// TIA Portal V17 export
// export: Created 2023-02-13T11:16:40.304202Z, ExportSetting WithDefaults, DisplayName Totally Integrated Automation Portal, DisplayVersion V17, DisplayName TIA Portal Openness, DisplayVersion V17, DisplayName TIA Portal Teamcenter Gateway, DisplayVersion V17, DisplayName TIA Portal Version Control Interface, DisplayVersion V17, DisplayName SINAMICS Startdrive Advanced, DisplayVersion V17, DisplayName SINAMICS Startdrive G130, G150, S120, S150, SINAMICS MV, S210, DisplayVersion V17, DisplayName SINAMICS Startdrive G110M, G120, G120C, G120D, G120P, G115D, DisplayVersion V17, DisplayName STEP 7 Professional, DisplayVersion V17, DisplayName STEP 7 Safety, DisplayVersion V17, DisplayName WinCC Professional, DisplayVersion V17
FUNCTION_BLOCK "Hot_Water"   // FB366, LAD
{ S7_Optimized_Access := 'TRUE' }
VERSION : 0.1
// stored: AutoNumber false, IsIECCheckEnabled false, IsRetainMemResEnabled false, MemoryReserve 100, SetENOAutomatically false, UDAEnableTagReadback false
   VAR_INPUT
      IN_FBAV_Inload : Bool;
      IN_FBAV_Outlet : Bool;
      IN_FBAV_Transfer : Bool;
      IN_FBP_Transfer : Bool;
      IN_FBP_Transfer_SP : Real;
      IN_Dose_Run : Bool;
      IN_Dose_Held : Bool;
      IN_Dose_Complete : Bool;
      IN_Dose_Header_1 : Bool;
      IN_Dose_Header_2 : Bool;
      IN_Dose_Valve_Cmd : Bool;
      IN_Dose_Pump_Cmd : Bool;
      IN_Dose_Pump_Sp : Real;
      IN_Dose_LineOK : Bool;
      IN_Low_Level : Bool;
      IN_Med_Level : Bool;
      IN_High_Level : Bool;
      IN_FBCV : Bool;
      "IN_FBCV_Act%" : Real;
      IN_Temperature : Real;
   END_VAR
   VAR_OUTPUT
      Out_AV_Inload : Bool;
      Out_AV_Outlet : Bool;
      Out_AV_Transfer : Bool;
      Out_P_Transfer : Bool;
      Out_P_Transfer_Sp : Real;
      OUT_CV : Bool;
      Out_Temp_Act : Real;
      Out_Temp_Sp : Real;
   END_VAR
   VAR
      Cmd : Struct
         Inload_Start : Bool;
         Inload_Mode : Bool := 1;   // 0 : Manual ;; 1 : Auto
         ReadyForTransfer : Bool;
         Transfer_Mode : Bool;   // 0 : By Timer ;; 1 : By Quantity
      END_STRUCT;
   END_VAR
   VAR RETAIN
      Param : Struct
         Temperature_SP : Real := 50.0;
      END_STRUCT;
   END_VAR
   VAR
      State : Struct
         Tank_LL : Bool;
         Tank_ML : Bool;
         Tank_HL : Bool;
         Inload_EN : Bool;
         Inload_Aut : Bool;
         Inloading : Bool;
         Ready_For_Transfer_EN : Bool;
         Ready_For_Transfer : Bool;
         Tank_Available : Bool;
         Transfer_on_Prog : Bool;
      END_STRUCT;
      alwaysON : Bool;
      r : Struct
         PosE1 : Bool;
         PosE2 : Bool;
         PosE3 : Bool;
         PosE4 : Bool;
         PosE5 : Bool;
         PosE6 : Bool;
         PosE7 : Bool;
         PosE8 : Bool;
         PosE9 : Bool;
         PosE10 : Bool;
         PosE11 : Bool;
         PosE12 : Bool;
         PosE13 : Bool;
         PosE14 : Bool;
         PosE15 : Bool;
         PosE16 : Bool;
         PosE17 : Bool;
         PosE18 : Bool;
         PosE19 : Bool;
         PosE20 : Bool;
         PosE21 : Bool;
         PosE22 : Bool;
         PosE23 : Bool;
         PosE24 : Bool;
         PosE25 : Bool;
         PosE26 : Bool;
         PosE27 : Bool;
         PosE28 : Bool;
         PosE29 : Bool;
         PosE30 : Bool;
         PosE31 : Bool;
         PosE32 : Bool;
      END_STRUCT;
      Actuator : Struct
         AV_Inload : Bool;
         AV_Outlet : Bool;
         AV_Transfer : Bool;
         AV_CIP_Tank : Bool;
         AV_CIP_Line : Bool;
         P_Transfer : Bool;
         P_Inload : Bool;
         P_CIP : Bool;
         CV : Bool;
      END_STRUCT;
      SPumpTim { S7_SetPoint := 'True'} : TON_TIME;
   END_VAR
   VAR_TEMP   // added for the SCL form of the ladder/FBD networks
      _w1 : Bool;
      _w2 : Bool;
   END_VAR
BEGIN

REGION Network 1: Always_ON
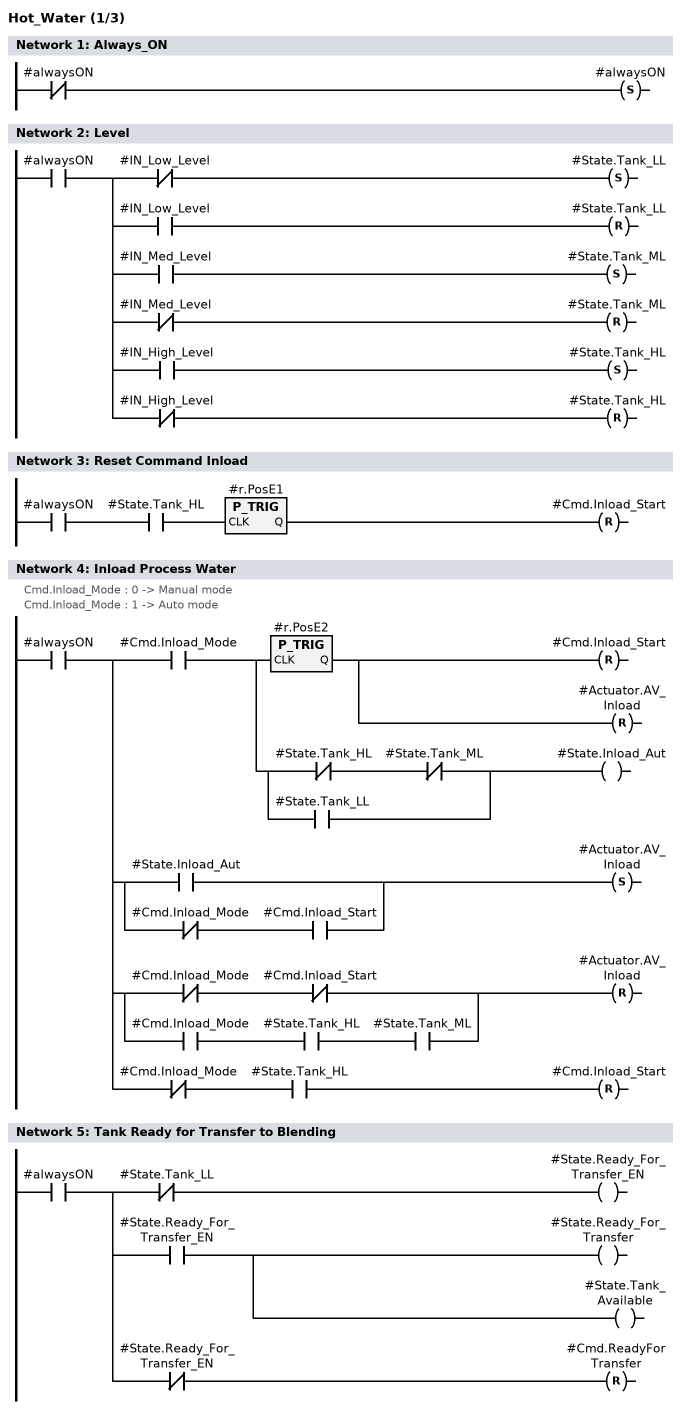
   RUNG wire#powerrail
      I_Contact( #alwaysON )
      S_Coil( #alwaysON )
   END_RUNG
   // the same network as SCL:
   IF NOT #alwaysON THEN #alwaysON := TRUE; END_IF;
END_REGION

REGION Network 2: Level
   RUNG wire#powerrail
      Contact( #alwaysON )
      wire#w1
      I_Contact( #IN_Low_Level )
      S_Coil( #State.Tank_LL )
   END_RUNG
   RUNG wire#w1
      Contact( #IN_Low_Level )
      R_Coil( #State.Tank_LL )
   END_RUNG
   RUNG wire#w1
      Contact( #IN_Med_Level )
      S_Coil( #State.Tank_ML )
   END_RUNG
   RUNG wire#w1
      I_Contact( #IN_Med_Level )
      R_Coil( #State.Tank_ML )
   END_RUNG
   RUNG wire#w1
      Contact( #IN_High_Level )
      S_Coil( #State.Tank_HL )
   END_RUNG
   RUNG wire#w1
      I_Contact( #IN_High_Level )
      R_Coil( #State.Tank_HL )
   END_RUNG
   // the same network as SCL:
   IF #alwaysON AND NOT #IN_Low_Level THEN #State.Tank_LL := TRUE; END_IF;
   IF #alwaysON AND #IN_Low_Level THEN #State.Tank_LL := FALSE; END_IF;
   IF #alwaysON AND #IN_Med_Level THEN #State.Tank_ML := TRUE; END_IF;
   IF #alwaysON AND NOT #IN_Med_Level THEN #State.Tank_ML := FALSE; END_IF;
   IF #alwaysON AND #IN_High_Level THEN #State.Tank_HL := TRUE; END_IF;
   IF #alwaysON AND NOT #IN_High_Level THEN #State.Tank_HL := FALSE; END_IF;
END_REGION

REGION Network 3: Reset Command Inload
   RUNG wire#powerrail
      Contact( #alwaysON )
      Contact( #State.Tank_HL )
      P_Trig( #r.PosE1 )
      R_Coil( #Cmd.Inload_Start )
   END_RUNG
   // the same network as SCL:
   #_w1 := #alwaysON AND #State.Tank_HL;
   #_w2 := #_w1 AND NOT #r.PosE1;   // rising edge
   #r.PosE1 := #_w1;
   IF #_w2 THEN #Cmd.Inload_Start := FALSE; END_IF;
END_REGION

REGION Network 4: Inload Process Water
   // Cmd.Inload_Mode : 0 -> Manual mode
   // Cmd.Inload_Mode : 1 -> Auto mode
   RUNG wire#powerrail
      Contact( #alwaysON )
      wire#w1
      Contact( #Cmd.Inload_Mode )
      wire#w2
      P_Trig( #r.PosE2 )
      wire#w3
      R_Coil( #Cmd.Inload_Start )
   END_RUNG
   RUNG wire#w3
      R_Coil( #Actuator.AV_Inload )
   END_RUNG
   RUNG wire#w2
      I_Contact( #State.Tank_HL )
      I_Contact( #State.Tank_ML )
      wire#w4
      Coil( #State.Inload_Aut )
   END_RUNG
   RUNG wire#w2
      Contact( #State.Tank_LL )
   END_RUNG wire#w4
   RUNG wire#w1
      Contact( #State.Inload_Aut )
      wire#w5
      S_Coil( #Actuator.AV_Inload )
   END_RUNG
   RUNG wire#w1
      I_Contact( #Cmd.Inload_Mode )
      Contact( #Cmd.Inload_Start )
   END_RUNG wire#w5
   RUNG wire#w1
      I_Contact( #Cmd.Inload_Mode )
      I_Contact( #Cmd.Inload_Start )
      wire#w6
      R_Coil( #Actuator.AV_Inload )
   END_RUNG
   RUNG wire#w1
      Contact( #Cmd.Inload_Mode )
      Contact( #State.Tank_HL )
      Contact( #State.Tank_ML )
   END_RUNG wire#w6
   RUNG wire#w1
      I_Contact( #Cmd.Inload_Mode )
      Contact( #State.Tank_HL )
      R_Coil( #Cmd.Inload_Start )
   END_RUNG
   // the same network as SCL:
   #_w1 := #alwaysON AND #Cmd.Inload_Mode;
   #_w2 := #_w1 AND NOT #r.PosE2;   // rising edge
   #r.PosE2 := #_w1;
   IF #_w2 THEN
       #Cmd.Inload_Start := FALSE;
       #Actuator.AV_Inload := FALSE;
   END_IF;
   #State.Inload_Aut := #_w1 AND ((NOT #State.Tank_HL AND NOT #State.Tank_ML) OR #State.Tank_LL);
   IF #alwaysON AND (#State.Inload_Aut OR (NOT #Cmd.Inload_Mode AND #Cmd.Inload_Start)) THEN
       #Actuator.AV_Inload := TRUE;
   END_IF;
   IF #alwaysON AND ((NOT #Cmd.Inload_Mode AND NOT #Cmd.Inload_Start) OR (#Cmd.Inload_Mode AND #State.Tank_HL AND #State.Tank_ML)) THEN
       #Actuator.AV_Inload := FALSE;
   END_IF;
   IF #alwaysON AND NOT #Cmd.Inload_Mode AND #State.Tank_HL THEN #Cmd.Inload_Start := FALSE; END_IF;
END_REGION

REGION Network 5: Tank Ready for Transfer to Blending
   RUNG wire#powerrail
      Contact( #alwaysON )
      wire#w1
      I_Contact( #State.Tank_LL )
      Coil( #State.Ready_For_Transfer_EN )
   END_RUNG
   RUNG wire#w1
      Contact( #State.Ready_For_Transfer_EN )
      wire#w2
      Coil( #State.Ready_For_Transfer )
   END_RUNG
   RUNG wire#w2
      Coil( #State.Tank_Available )
   END_RUNG
   RUNG wire#w1
      I_Contact( #State.Ready_For_Transfer_EN )
      R_Coil( #Cmd.ReadyForTransfer )
   END_RUNG
   // the same network as SCL:
   #State.Ready_For_Transfer_EN := #alwaysON AND NOT #State.Tank_LL;
   #State.Ready_For_Transfer := #alwaysON AND #State.Ready_For_Transfer_EN;
   #State.Tank_Available := #State.Ready_For_Transfer;
   IF #alwaysON AND NOT #State.Ready_For_Transfer_EN THEN #Cmd.ReadyForTransfer := FALSE; END_IF;
END_REGION

REGION Network 6: Transfer to Blending AV and Pump
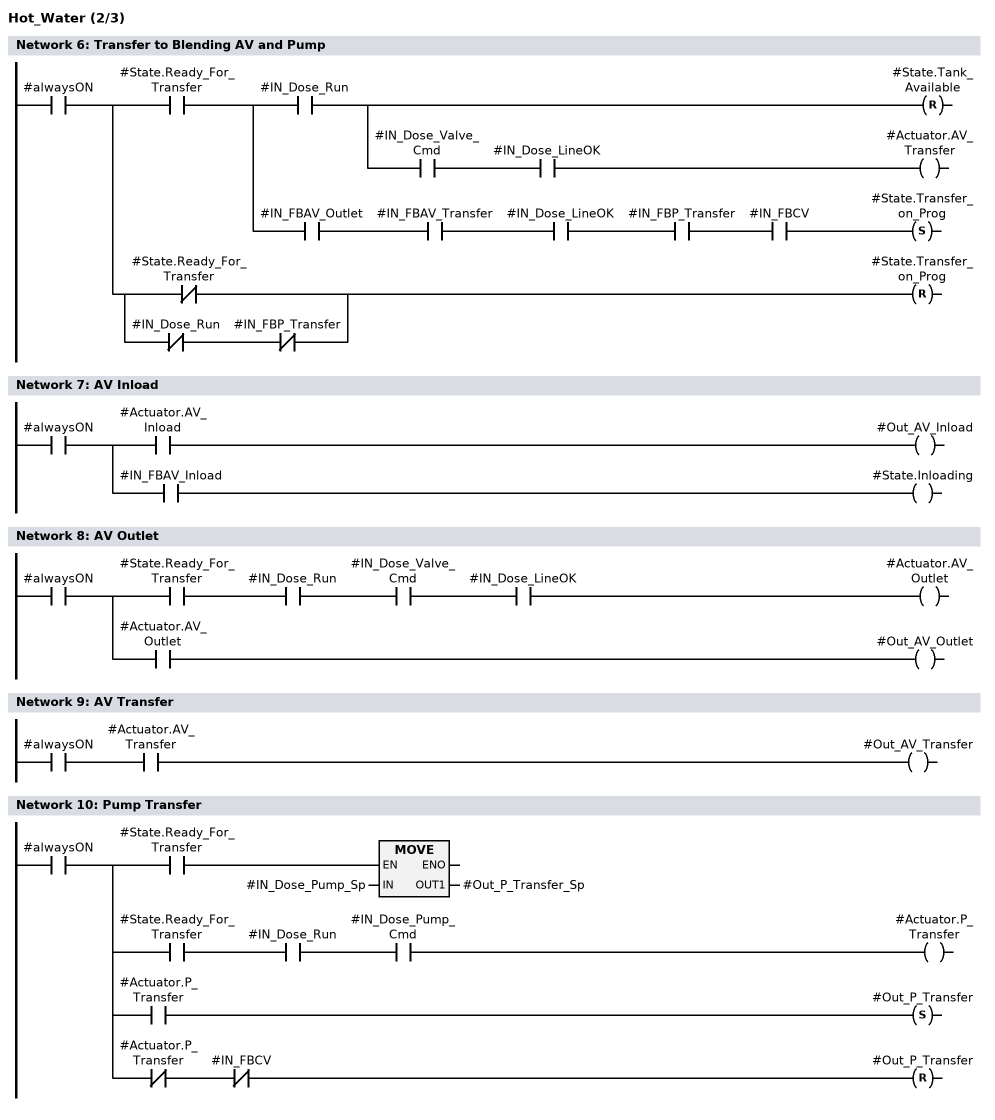
   RUNG wire#powerrail
      Contact( #alwaysON )
      wire#w1
      Contact( #State.Ready_For_Transfer )
      wire#w2
      Contact( #IN_Dose_Run )
      wire#w3
      R_Coil( #State.Tank_Available )
   END_RUNG
   RUNG wire#w3
      Contact( #IN_Dose_Valve_Cmd )
      Contact( #IN_Dose_LineOK )
      Coil( #Actuator.AV_Transfer )
   END_RUNG
   RUNG wire#w2
      Contact( #IN_FBAV_Outlet )
      Contact( #IN_FBAV_Transfer )
      Contact( #IN_Dose_LineOK )
      Contact( #IN_FBP_Transfer )
      Contact( #IN_FBCV )
      S_Coil( #State.Transfer_on_Prog )
   END_RUNG
   RUNG wire#w1
      I_Contact( #State.Ready_For_Transfer )
      wire#w4
      R_Coil( #State.Transfer_on_Prog )
   END_RUNG
   RUNG wire#w1
      I_Contact( #IN_Dose_Run )
      I_Contact( #IN_FBP_Transfer )
   END_RUNG wire#w4
   // the same network as SCL:
   #_w1 := #alwaysON AND #State.Ready_For_Transfer;
   #_w2 := #_w1 AND #IN_Dose_Run;
   IF #_w2 THEN #State.Tank_Available := FALSE; END_IF;
   #Actuator.AV_Transfer := #_w2 AND #IN_Dose_Valve_Cmd AND #IN_Dose_LineOK;
   IF #_w1 AND #IN_FBAV_Outlet AND #IN_FBAV_Transfer AND #IN_Dose_LineOK AND #IN_FBP_Transfer AND #IN_FBCV THEN
       #State.Transfer_on_Prog := TRUE;
   END_IF;
   IF #alwaysON AND (NOT #State.Ready_For_Transfer OR (NOT #IN_Dose_Run AND NOT #IN_FBP_Transfer)) THEN
       #State.Transfer_on_Prog := FALSE;
   END_IF;
END_REGION

REGION Network 7: AV Inload
   RUNG wire#powerrail
      Contact( #alwaysON )
      wire#w1
      Contact( #Actuator.AV_Inload )
      Coil( #Out_AV_Inload )
   END_RUNG
   RUNG wire#w1
      Contact( #IN_FBAV_Inload )
      Coil( #State.Inloading )
   END_RUNG
   // the same network as SCL:
   #Out_AV_Inload := #alwaysON AND #Actuator.AV_Inload;
   #State.Inloading := #alwaysON AND #IN_FBAV_Inload;
END_REGION

REGION Network 8: AV Outlet
   RUNG wire#powerrail
      Contact( #alwaysON )
      wire#w1
      Contact( #State.Ready_For_Transfer )
      Contact( #IN_Dose_Run )
      Contact( #IN_Dose_Valve_Cmd )
      Contact( #IN_Dose_LineOK )
      Coil( #Actuator.AV_Outlet )
   END_RUNG
   RUNG wire#w1
      Contact( #Actuator.AV_Outlet )
      Coil( #Out_AV_Outlet )
   END_RUNG
   // the same network as SCL:
   #Actuator.AV_Outlet := #alwaysON AND #State.Ready_For_Transfer AND #IN_Dose_Run AND #IN_Dose_Valve_Cmd AND #IN_Dose_LineOK;
   #Out_AV_Outlet := #alwaysON AND #Actuator.AV_Outlet;
END_REGION

REGION Network 9: AV Transfer
   RUNG wire#powerrail
      Contact( #alwaysON )
      Contact( #Actuator.AV_Transfer )
      Coil( #Out_AV_Transfer )
   END_RUNG
   // the same network as SCL:
   #Out_AV_Transfer := #alwaysON AND #Actuator.AV_Transfer;
END_REGION

REGION Network 10: Pump Transfer
   RUNG wire#powerrail
      Contact( #alwaysON )
      wire#w1
      Contact( #State.Ready_For_Transfer )
      Move(in := #IN_Dose_Pump_Sp, out1 => #Out_P_Transfer_Sp)
   END_RUNG
   RUNG wire#w1
      Contact( #State.Ready_For_Transfer )
      Contact( #IN_Dose_Run )
      Contact( #IN_Dose_Pump_Cmd )
      Coil( #Actuator.P_Transfer )
   END_RUNG
   RUNG wire#w1
      Contact( #Actuator.P_Transfer )
      S_Coil( #Out_P_Transfer )
   END_RUNG
   RUNG wire#w1
      I_Contact( #Actuator.P_Transfer )
      I_Contact( #IN_FBCV )
      R_Coil( #Out_P_Transfer )
   END_RUNG
   // the same network as SCL:
   IF #alwaysON AND #State.Ready_For_Transfer THEN #Out_P_Transfer_Sp := #IN_Dose_Pump_Sp; END_IF;
   #Actuator.P_Transfer := #alwaysON AND #State.Ready_For_Transfer AND #IN_Dose_Run AND #IN_Dose_Pump_Cmd;
   IF #alwaysON AND #Actuator.P_Transfer THEN #Out_P_Transfer := TRUE; END_IF;
   IF #alwaysON AND NOT #Actuator.P_Transfer AND NOT #IN_FBCV THEN #Out_P_Transfer := FALSE; END_IF;
END_REGION

REGION Network 11: Control Valve
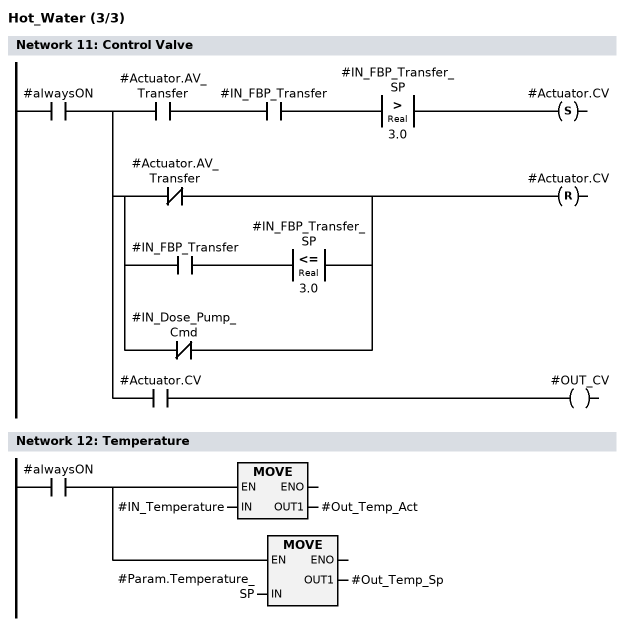
   RUNG wire#powerrail
      Contact( #alwaysON )
      wire#w1
      Contact( #Actuator.AV_Transfer )
      Contact( #IN_FBP_Transfer )
      { S7_Templates := "SrcType := Real" } GT_Contact(in1 := #IN_FBP_Transfer_SP, in2 := 3.0)
      S_Coil( #Actuator.CV )
   END_RUNG
   RUNG wire#w1
      I_Contact( #Actuator.AV_Transfer )
      wire#w2
      R_Coil( #Actuator.CV )
   END_RUNG
   RUNG wire#w1
      Contact( #IN_FBP_Transfer )
      { S7_Templates := "SrcType := Real" } LE_Contact(in1 := #IN_FBP_Transfer_SP, in2 := 3.0)
   END_RUNG wire#w2
   RUNG wire#w1
      I_Contact( #IN_Dose_Pump_Cmd )
   END_RUNG wire#w2
   RUNG wire#w1
      Contact( #Actuator.CV )
      Coil( #OUT_CV )
   END_RUNG
   // the same network as SCL:
   IF #alwaysON AND #Actuator.AV_Transfer AND #IN_FBP_Transfer AND (#IN_FBP_Transfer_SP > 3.0) THEN
       #Actuator.CV := TRUE;
   END_IF;
   IF #alwaysON AND (NOT #Actuator.AV_Transfer OR (#IN_FBP_Transfer AND (#IN_FBP_Transfer_SP <= 3.0)) OR NOT #IN_Dose_Pump_Cmd) THEN
       #Actuator.CV := FALSE;
   END_IF;
   #OUT_CV := #alwaysON AND #Actuator.CV;
END_REGION

REGION Network 12: Temperature
   RUNG wire#powerrail
      Contact( #alwaysON )
      wire#w1
      Move(in := #IN_Temperature, out1 => #Out_Temp_Act)
   END_RUNG
   RUNG wire#w1
      Move(in := #Param.Temperature_SP, out1 => #Out_Temp_Sp)
   END_RUNG
   // the same network as SCL:
   IF #alwaysON THEN
       #Out_Temp_Act := #IN_Temperature;
       #Out_Temp_Sp := #Param.Temperature_SP;
   END_IF;
END_REGION
END_FUNCTION_BLOCK
